(* IEC 61131-3 sources: test/Class/AI046 (part 2) *)

//**********************************************************************************************************************************************************
  ELSE
    // we forward this message to the base class
		ret_code := SdiasBase::NewInst(pPara, pResult);
	END_CASE;

END_FUNCTION
